FUNCTION_BLOCK Test_TStreamAdd_Read_UDINT EXTENDS T_UnitTestBase
VAR
    Stream  : T_Stream(StreamLength := 2);
    ArgType : E_ArgTypeId := E_ArgTypeId.Type_UDINT;
END_VAR

{attribute 'analysis' := '-33'} // inhibit unused variable warning
METHOD RunTest
Stream.Init(2);

// add a UDINT...
Stream.SetNextArgTypeId(ArgType);
Stream.Add_UDINT(12345678);

Stream.SetReadPosition(0);

// check next arg type is correct...
AssertEquals_INT(Expected     := ArgType,
                           Actual       := Stream.GetNextArgTypeId(),
                           Message := 'Stream.GetNextArgTypeId()');

// check next value...	
AssertEquals_UDINT(Expected     := 12345678,
                             Actual       := Stream.Read_UDINT(),
                             Message := 'Stream.Read_UDINT()');

// check we are at the end of the stream..							
AssertEquals_UDINT(Expected     := Stream.StreamLength,
                             Actual       := Stream.ReadPosition,
                             Message := 'Stream.ReadPosition');

TestCompleted := TRUE;
END_METHOD

END_FUNCTION_BLOCK

(* stored: Version 1.1.0.1, ProductVersion 3.1.4024.12
   POU Test_TStreamAdd_Read_UDINT: Id {98133168-3ecc-4528-8e23-6c4f325cb3e7}, SpecialFunc None
   Method RunTest: Id {51b97a74-e859-4c85-925e-a18affe75f1b} *)
